(* IEC 61131-3 sources: generating_plc_code_with_llms/Code#2/ChatGPT_3.5/second run, 21 files *)

(* ---- 14.st ---- *)
// 7.18s
// 2
FUNCTION FC1001 :BOOL
VAR_INPUT
    MEW: REAL;
    SP: REAL;
    HYS: REAL;
END_VAR
VAR_IN_OUT
    OUT:BOOL;
END_VAR
VAR
    P_HYS: REAL;
END_VAR
    // Calculate the switching hysteresis as a percentage of the setpoint
    P_HYS := SP * HYS / 100.0;

    // Check if the measured value exceeds the upper threshold
    IF MEW > SP + P_HYS THEN
        OUT := TRUE;
    ELSIF MEW < SP - P_HYS THEN
        OUT := FALSE;
    END_IF;

    // Return the output status
    RETURN OUT;
END_FUNCTION

(* ---- 15.st ---- *)
// 8.77s
// 2
FUNCTION FC1002 :BOOL
VAR_INPUT
    E_A, SENSOR: BOOL;
    ZEITW: TIME;
END_VAR
VAR_IN_OUT
    ZEIT:TON;
    P_HU, P_AL: BOOL;
END_VAR
    // Check if the monitoring system is switched on
    IF E_A THEN
        // Reset the timer if the sensor reports an approach
        IF SENSOR THEN
            ZEIT(IN := FALSE);
        ELSE
            // Start the timer if the sensor doesn't report an approach
            ZEIT(IN := TRUE, PT := ZEITW);
        END_IF;

        // Check if the timer has reached the specified time
        IF ZEIT.Q THEN
            // Switch off the warning signal and turn on the alarm
            P_HU := FALSE;
            P_AL := TRUE;
        ELSE
            // Switch on the warning signal
            P_HU := SENSOR;
            // Turn off the alarm
            P_AL := FALSE;
        END_IF;
    ELSE
        // Switch off the monitoring system, warning signal, and alarm
        ZEIT(IN := FALSE);
        P_HU := FALSE;
        P_AL := FALSE;
    END_IF;

    // Return the switched on status of the monitoring system
    RETURN E_A;
END_FUNCTION

(* ---- 18.st ---- *)
// 6.77s
// 4
FUNCTION FC1003 : VOID
VAR_INPUT
    IN_R: REAL;
    IN_MAX, IN_MIN: REAL;
    OUT_MAX, OUT_MIN: REAL;
END_VAR
VAR_OUTPUT
    OUT_R: REAL;
    FEH: BOOL;
END_VAR
VAR_TEMP
    DIFF1, DIFF2: REAL;
END_VAR

IF (IN_MAX <> IN_MIN) THEN
    // Calculate the difference between the input and output ranges
    DIFF1 := OUT_MAX - OUT_MIN;
    DIFF2 := IN_MAX - IN_MIN;

    // Perform the range mapping
    OUT_R := OUT_MIN + ((IN_R - IN_MIN) / DIFF2) * DIFF1;

    // Check for out-of-range conditions
    IF (OUT_R < OUT_MIN) THEN
        OUT_R := OUT_MIN;
        FEH := TRUE;  // Set error flag
    ELSIF (OUT_R > OUT_MAX) THEN
        OUT_R := OUT_MAX;
        FEH := TRUE;  // Set error flag
    ELSE
        FEH := FALSE; // No error
    END_IF;
ELSE
    // Avoid division by zero if IN_MAX is equal to IN_MIN
    OUT_R := OUT_MIN;
    FEH := TRUE;  // Set error flag
END_IF;

(* ---- 19.st ---- *)
// 11.44s
// 2
FUNCTION_BLOCK FB1005
VAR_INPUT
    START: BOOL;
    DICKE, V_MAX, V_MIN: REAL;
END_VAR
VAR_OUTPUT
    D_MAX, D_MIN: REAL;
    P1: BOOL;
END_VAR
VAR
    FO: BOOL;
    M_MAX, M_MIN: REAL;
END_VAR
METHOD Messung : BOOL
    // Measure the thickness and update M_MAX, M_MIN
    M_MAX := MAX(M_MAX, DICKE);
    M_MIN := MIN(M_MIN, DICKE);

    // Check if the measured values are outside the tolerance band
    IF M_MAX > V_MAX OR M_MIN < V_MIN THEN
        P1 := TRUE;  // Turn on the reject light
    ELSE
        P1 := FALSE; // Turn off the reject light
    END_IF;

    // Return FALSE to end the measurement
    RETURN FALSE;
END_METHOD

METHOD StartMeasurement : BOOL
    // Start a new measurement cycle
    M_MAX := 0;
    M_MIN := 0;
    P1 := FALSE; // Turn off the reject light

    // Return TRUE to start the measurement
    RETURN TRUE;
END_METHOD

METHOD EndMeasurement : BOOL
    // Update output values with the results of the measurement
    D_MAX := M_MAX;
    D_MIN := M_MIN;

    // Return FALSE to end the measurement
    RETURN FALSE;
END_METHOD

METHOD FB1005 : BOOL
    // Check if the measurement is ongoing
    IF START THEN
        // If not in the measurement, start a new cycle
        IF NOT FO THEN
            FO := TRUE;
            RETURN StartMeasurement();
        // If already in the measurement, continue
        ELSE
            RETURN Messung();
        END_IF;
    // If the sensor is off, end the measurement
    ELSE
        IF FO THEN
            FO := FALSE;
            RETURN EndMeasurement();
        END_IF;
    END_IF;
END_METHOD
END_FUNCTION_BLOCK

(* ---- 20.st ---- *)
// 10.46s
// 2
FUNCTION_BLOCK INTERLOCK
VAR_INPUT
    I1: BOOL;
    I2: BOOL;
    TL: TIME;
END_VAR
VAR_OUTPUT
    Q1: BOOL;
    Q2: BOOL;
END_VAR
VAR
    T1: TOF;
    T2: TOF;
END_VAR

METHOD InterlockControl: BOOL
    // Control the interlock logic
    IF NOT T1.PT THEN
        // Start timer T1 when I1 is TRUE
        T1(IN := I1, PT := TL);
    ELSE
        // Reset timer T1 when I1 goes FALSE
        T1(IN := NOT I1);
    END_IF;

    IF NOT T2.PT THEN
        // Start timer T2 when I2 is TRUE
        T2(IN := I2, PT := TL);
    ELSE
        // Reset timer T2 when I2 goes FALSE
        T2(IN := NOT I2);
    END_IF;

    // Set Q1 only if T1 is not running and I1 is TRUE
    IF NOT T1.Q THEN
        Q1 := I1;
    END_IF;

    // Set Q2 only if T2 is not running and I2 is TRUE
    IF NOT T2.Q THEN
        Q2 := I2;
    END_IF;

    // Return TRUE to keep the method running
    RETURN TRUE;
END_METHOD

METHOD Initialize: BOOL
    // Reset timers and outputs at the beginning
    T1(IN := FALSE);
    T2(IN := FALSE);
    Q1 := FALSE;
    Q2 := FALSE;

    // Return FALSE to end the initialization
    RETURN FALSE;
END_METHOD

METHOD INTERLOCK: BOOL
    // Run the initialization at the start
    IF NOT T1.Q THEN
        RETURN Initialize();
    ELSE
        // Run the interlock control logic
        RETURN InterlockControl();
    END_IF;
END_METHOD
END_FUNCTION_BLOCK

(* ---- 21.st ---- *)
// 47.04s
// weiter generieren
// 2
FUNCTION_BLOCK BURNER
VAR_INPUT
    IN : BOOL;
    STAGE2 : BOOL;
    OVER_TEMP : BOOL;
    OIL_TEMP : BOOL := TRUE;
    FLAME : BOOL;
    RST : BOOL;
    RST_TIMER : BOOL;
    PRE_HEAT_TIME : TIME := t#5s;
    PRE_VENT_TIME : TIME := t#15s;
    PRE_IGNITE_TIME : TIME := t#15s;
    POST_IGNITE_TIME : TIME := t#25s;
    STAGE2_DELAY : TIME := t#10s;
    SAFETY_TIME : TIME := t#5s;
    LOCKOUT_TIME : TIME := t#10s;
    MULTIPLE_IGNITION : BOOL := TRUE;
    KW1 : REAL;
    KW2 : REAL;
END_VAR
VAR_OUTPUT
    MOTOR : BOOL;
    COIL1 : BOOL;
    COIL2 : BOOL;
    PRE_HEAT : BOOL;
    IGNITE : BOOL;
    FAIL : BOOL;
    KWH : REAL;
    STATUS : BYTE;
END_VAR
VAR_IN_OUT
    RUNTIME1 : UDINT;
    RUNTIME2 : UDINT;
    CYCLES : UDINT;
END_VAR
VAR
    state : INT;
    last : TIME;
    tx : TIME;
    last_change : TIME;
    timer1 : TON;
    timer2 : TON;
    oil_temp_last : BOOL;
    cycles2 : UDINT;
END_VAR

METHOD BurnerControl : BOOL
    tx := Tcyclic - last;
    last := Tcyclic;

    // Reset error flags
    FAIL := FALSE;

    // State machine for burner control
    CASE state OF
        110:
            // Standby - Wait for start signal
            IF IN THEN
                PRE_HEAT := TRUE;
                state := 111;  // Transition to startup sequence
            END_IF;
        111:
            // Startup Sequence
            IF (NOT OVER_TEMP) AND (NOT PRE_HEAT) THEN
                // Continue with startup sequence
                IF NOT OIL_TEMP THEN
                    IF timer1(IN := TRUE, PT := PRE_HEAT_TIME) THEN
                        // Fuel oil warming has not responded in time
                        STATUS := 1;
                        FAIL := TRUE;
                        state := 110;  // Return to standby
                    END_IF;
                ELSE
                    // Fuel oil warming responded, move to next step
                    MOTOR := TRUE;
                    COIL1 := TRUE;
                    timer1(IN := TRUE, PT := PRE_VENT_TIME);
                    state := 112;
                END_IF;
            END_IF;
        112:
            // Burner runs on stage 1
            IF timer1.Q THEN
                IGNITE := TRUE;
                COIL1 := FALSE;
                timer2(IN := TRUE, PT := PRE_IGNITE_TIME);
                state := 113;
            END_IF;
        113:
            // Burner runs on stage 2
            IF (STAGE2 AND timer2.Q) THEN
                COIL2 := TRUE;
            END_IF;
    END_CASE;

    // Check for errors during startup sequence
    IF (state = 112) AND FLAME THEN
        // Flame sensor is active during aeration
        STATUS := 2;
        FAIL := TRUE;
        state := 110;  // Return to standby
    END_IF;

    // Check for errors during burner operation
    IF (state = 113) AND (NOT FLAME) THEN
        IF timer2.Q THEN
            // No flame after specified time
            STATUS := 4;
            FAIL := TRUE;
            state := 110;  // Return to standby
        END_IF;

        // Check for multiple ignitions
        IF MULTIPLE_IGNITION AND FLAME AND (timer2.ET > 0) THEN
            IGNITE := TRUE;
            COIL2 := FALSE;
            cycles2 := cycles2 + 1;
            state := 113;
        END_IF;
    END_IF;

    // Boiler overheating protection
    IF OVER_TEMP THEN
        STATUS := 9;
        FAIL := TRUE;
        state := 110;  // Return to standby
    END_IF;

    // Lockout timer
    IF FAIL THEN
        IF NOT RST_TIMER THEN
            IF timer1.Q OR timer2.Q THEN
                timer1(IN := FALSE);
                timer2(IN := FALSE);
                timer1(IN := FALSE, PT := LOCKOUT_TIME);
                state := 110;  // Return to standby
            END_IF;
        END_IF;
    END_IF;

    // Update runtime and cycles
    IF state = 113 THEN
        RUNTIME1 := RUNTIME1 + tx;
    END_IF;

    // Update outputs
    KWH := (REAL)(cycles2 + (state = 113)) * KW2 + (REAL)CYCLES * KW1;
    CYCLES := cycles2 + (state = 113);

    RETURN state = 113;  // Return TRUE when the burner is running
END_METHOD;

METHOD BurnerStatus : VOID
    // Output the current status
    CASE state OF
        110: STATUS := 110;  // Standby
        111: STATUS := 111;  // Startup sequence is executed
        112: STATUS := 112;  // Burner runs on stage 1
        113: STATUS := 113;  // Burner runs on stage 2
    END_CASE;
END_METHOD;
END_FUNCTION_BLOCK

(* ---- 1.st ---- *)
// 4.91s
// 3
VAR
    xAllOn : BOOL;
    xAllOff : BOOL;

    xAlarm1 : BOOL;
    xAlarm2 : BOOL;
END_VAR

xAllOn := FALSE;
xAllOff := FALSE;
xAlarm1 := FALSE;
xAlarm2 := FALSE;

IF xAllOn THEN
    xAlarm1 := TRUE;
    xAlarm2 := TRUE;
    xAllOn := FALSE;
END_IF

IF xAllOff THEN
    xAlarm1 := FALSE;
    xAlarm2 := FALSE;
    xAllOff := FALSE;
END_IF

(* ---- 10.st ---- *)
// 4.44s
// 4
VAR_INPUT
    X : REAL;
END_VAR

VAR
    Y : REAL;
END_VAR

Y := 1 / (1 + EXP(-X));

(* ---- 11.st ---- *)
// 4.02s
// 4
VAR_INPUT
    x : REAL;
END_VAR

VAR
    result : INT;
END_VAR

IF x > 0 THEN
    result := 1;
ELSIF x < 0 THEN
    result := -1;
ELSE
    result := 0;
END_IF

(* ---- 12.st ---- *)
// 4.07s
// 4
VAR
    X : REAL;
    sinhX : REAL;
END_VAR

sinhX := (EXP(X) - EXP(-X)) / 2.0;

(* ---- 13.st ---- *)
// 5.81s
// 2
VAR CONSTANT
    MAXNUMBERS : UINT := 99;
END_VAR

VAR
    aNumbers : ARRAY[0..MAXNUMBERS] OF INT;
    nCnt : INT;
END_VAR

nCnt := 0;

REPEAT
    // Check if the current number is 10
    IF aNumbers[nCnt] = 10 THEN
        // Abort the search if 10 is found
        EXIT;
    END_IF;

    // Increment the counter
    nCnt := nCnt + 1;

    // Check if the end of the list is reached
    IF nCnt > MAXNUMBERS THEN
        // Abort if the end of the list is reached without finding 10
        EXIT;
    END_IF;
UNTIL FALSE;

(* ---- 16.st ---- *)
// 10.51s
// 2
VAR
    North_green : BOOL;
    North_yellow : BOOL;
    North_red : BOOL;
    East_green : BOOL;
    East_yellow : BOOL;
    East_red : BOOL;
    T1 : TON;
END_VAR

T1(IN := TRUE, PT := T#5000ms);  // Timer T1 for the overall cycle

IF T1.Q THEN
    // Between 0ms and 5000ms
    North_green := TRUE;
    North_yellow := FALSE;
    North_red := FALSE;
    East_green := FALSE;
    East_yellow := FALSE;
    East_red := TRUE;
ELSE
    // After 5000ms
    North_green := FALSE;
    North_yellow := TRUE;
    North_red := FALSE;
    East_green := FALSE;
    East_yellow := FALSE;
    East_red := TRUE;
END_IF;

IF NOT T1.Q AND T1.ET THEN
    // Between 5500ms and 9500ms
    North_green := FALSE;
    North_yellow := FALSE;
    North_red := TRUE;
    East_green := TRUE;
    East_yellow := FALSE;
    East_red := FALSE;
END_IF;

IF NOT T1.Q AND T1.ETT THEN
    // Between 9500ms and 10000ms
    North_green := FALSE;
    North_yellow := FALSE;
    North_red := TRUE;
    East_green := FALSE;
    East_yellow := TRUE;
    East_red := FALSE;
END_IF;

(* ---- 17.st ---- *)
// 7.22s
// 4
VAR
    aiOutside : INT;
    aiHumidity: INT;
    sShowText : STRING[80];
END_VAR

// Read temperature and humidity values (replace with actual input values)
aiOutside := ...;
aiHumidity := ...;

// Evaluate temperature
IF aiOutside < 18 THEN
    sShowText := 'Cold';
ELSIF aiOutside >= 18 AND aiOutside <= 25 THEN
    // Evaluate humidity within the nested IF
    IF aiHumidity >= 40 AND aiHumidity <= 75 THEN
        sShowText := 'Opt';
    ELSE
        sShowText := 'Temp. OK';
    END_IF;
ELSE
    sShowText := 'Hot';
END_IF;

(* ---- 2.st ---- *)
// 4.61s
// 4
VAR_INPUT
    N : INT;
    K : INT;
    i : INT;
END_VAR

VAR
    result : INT;
    numerator : INT;
    denominator : INT;
END_VAR

result := 0;
numerator := 1;
denominator := 1;

IF K >= 0 AND K <= N THEN
    FOR i := 1 TO K DO
        numerator := numerator * (N - i + 1);
        denominator := denominator * i;
    END_FOR

    result := numerator / denominator;
END_IF

(* ---- 3.st ---- *)
// 4.94s
// 2
VAR_INPUT
    X : INT;
END_VAR

VAR
    t1 : DINT;
    t2 : DINT;
    x_tmp : INT;
END_VAR

t1 := 0;
t2 := 1;

IF X = 0 THEN
    x_tmp := t1;
ELSIF X = 1 THEN
    x_tmp := t2;
ELSE
    FOR i := 2 TO X DO
        x_tmp := t1 + t2;
        t1 := t2;
        t2 := x_tmp;
    END_FOR
END_IF

(* ---- 4.st ---- *)
// 7.06s
// 2
VAR
    aiLevel : INT;
    PercentLevel : UINT;
    doLow : BOOL;
    doOk : BOOL;
    doHigh : BOOL;
    doAlarm : BOOL;
END_VAR

aiLevel := ... // Read the analog input level (0 - 32767) from your system

// Convert analog input to percentage (0 - 100%)
PercentLevel := UINT_TO(aiLevel * 100 / 32767);

CASE PercentLevel OF
    (PercentLevel < 1):
        doLow := TRUE;
        doOk := FALSE;
        doHigh := FALSE;
        doAlarm := TRUE; // Activate the warning horn
    (PercentLevel >= 1 AND PercentLevel <= 75):
        doLow := FALSE;
        doOk := TRUE;
        doHigh := FALSE;
        doAlarm := FALSE;
    (PercentLevel > 75):
        doLow := FALSE;
        doOk := FALSE;
        doHigh := TRUE;
        doAlarm := FALSE;
END_CASE

(* ---- 5.st ---- *)
// 7.51s
// 3
VAR
    Start_Loop : BOOL := FALSE;
    one_hour : TIME := T#1h;
    One_Hour_Timer : TON;
    Gate_Open : BOOL := FALSE;
    Close_Gate_Inst : BOOL := FALSE;
    Sensed_Car : BOOL := FALSE;
    Sensed_Car_Inst : BOOL := FALSE;
    Sensed_App : BOOL := FALSE;
    Mobile_Inst : BOOL := FALSE;
    Auth : STRING;
    my_defined_str : STRING := 'abcd';
END_VAR

// Main control logic
IF NOT Start_Loop THEN
    // Start the one-hour timer when Start_Loop is FALSE
    One_Hour_Timer(IN := NOT Gate_Open AND NOT Close_Gate_Inst, PT := one_hour);

    // Check if the timer timed out
    IF One_Hour_Timer.Q THEN
        Close_Gate_Inst := TRUE;
    END_IF;

    // Check for sensed car or app with matching Auth string
    IF (Sensed_Car AND NOT Sensed_Car_Inst) OR (Sensed_App AND Mobile_Inst AND Auth = my_defined_str) THEN
        Gate_Open := TRUE;
        Close_Gate_Inst := FALSE;
    END_IF;

    // Reset the timer if the gate is open
    IF Gate_Open THEN
        One_Hour_Timer(IN := FALSE);
    END_IF;
ELSE
    // Reset the timer when Start_Loop is TRUE
    One_Hour_Timer(IN := FALSE);
    Close_Gate_Inst := FALSE;
    Gate_Open := FALSE;
END_IF

(* ---- 6.st ---- *)
// 12.6s
// 4
VAR CONSTANT
    WAIT : UINT:= 0;
    TOP_POSITION : UINT:= 1;
    BOTTOM_POSITION : UINT:= 2;
    GETBOX : UINT:= 3;
    UNLOAD_POSITION : UINT:= 4;
    UNLOAD_BOX : UINT:= 5;
END_VAR

VAR
    doConvTop: BOOL;
    doConvBottom: BOOL;
    doConvLift: BOOL;
    doLiftTop: BOOL;
    doLiftBottom: BOOL;
    doLiftUnload: BOOL;
    diConvTop: BOOL;
    diConvBottom: BOOL;
    diLiftTop: BOOL;
    diLiftBottom: BOOL;
    diLiftUnload: BOOL;
    diBoxLift: BOOL;
    selectLift: UINT;
    ConvTopOn: BOOL;
    ConvBottomOn: BOOL;
END_VAR

CASE selectLift OF
    WAIT:
        // Check if either light barrier is activated
        IF diConvTop THEN
            doConvTop := FALSE;
            ConvTopOn := FALSE;
            selectLift := TOP_POSITION;
        ELSIF diConvBottom THEN
            doConvBottom := FALSE;
            ConvBottomOn := FALSE;
            selectLift := BOTTOM_POSITION;
        END_IF;
        // Reset lift control signals
        doLiftTop := FALSE;
        doLiftBottom := FALSE;
        doLiftUnload := FALSE;
    TOP_POSITION:
        // Move lift to top position
        doLiftTop := TRUE;
        IF diLiftTop THEN
            doLiftTop := FALSE;
            selectLift := GETBOX;
        END_IF;
    BOTTOM_POSITION:
        // Move lift to bottom position
        doLiftBottom := TRUE;
        IF diLiftBottom THEN
            doLiftBottom := FALSE;
            selectLift := GETBOX;
        END_IF;
    GETBOX:
        // Activate lift conveyor until crate is at lift
        doConvLift := TRUE;
        IF diBoxLift THEN
            doConvLift := FALSE;
            selectLift := UNLOAD_POSITION;
        END_IF;
    UNLOAD_POSITION:
        // Move lift to unload position
        doLiftUnload := TRUE;
        IF diLiftUnload THEN
            doLiftUnload := FALSE;
            selectLift := UNLOAD_BOX;
        END_IF;
    UNLOAD_BOX:
        // Unload box onto the unloading conveyor
        // Once the box has left the lift, it's ready for the next request
        IF NOT diBoxLift THEN
            selectLift := WAIT;
        END_IF;
END_CASE;

(* ---- 7.st ---- *)
// 5.63s
// 2
VAR CONSTANT
    MAX_INDEX: USINT := 4;
END_VAR

VAR
    aWeights : ARRAY[0..MAX_INDEX] OF INT;
    iCnt : USINT;
    sumWeight : DINT;
    avgWeight : INT;
END_VAR

sumWeight := 0;

FOR iCnt := 0 TO MAX_INDEX DO
    // Read individual loads from analog inputs (replace with actual input values)
    aWeights[iCnt] := ...;
    sumWeight := sumWeight + aWeights[iCnt];
END_FOR

// Calculate average weight
IF MAX_INDEX > 0 THEN
    avgWeight := sumWeight / (MAX_INDEX + 1);
ELSE
    avgWeight := 0; // To avoid division by zero
END_IF

(* ---- 8.st ---- *)
// 7.08s
// 2
VAR_INPUT
    X : REAL;
END_VAR

VAR
    w : REAL;
    i : INT;
    we : REAL;
    w1e : REAL;
    ewx : REAL;
    last : DWORD;
END_VAR

w := 0.0;
i := 0;
we := 0.0;
w1e := 0.0;

FOR i := 0 TO 1000 DO
    ewx := EXP(w * we);
    last := TIME();
    w := w - (w * we - X) / (we * (w + 1));
    IF ABS(ewx - EXP(w * we)) < 1.0E-9 OR ABS(TIME() - last) < T#1ms THEN
        EXIT; // Exit loop if convergence or max iterations reached
    END_IF;
END_FOR

(* ---- 9.st ---- *)
// 5.72s
// 2
VAR
    YEAR : INT;
END_VAR

IF (YEAR MOD 4 = 0 AND YEAR MOD 100 <> 0) OR (YEAR MOD 400 = 0) THEN
    // Leap year conditions:
    // - If divisible by 4 but not by 100
    // - If divisible by 400
    // It is a leap year
    // Implement your logic for a leap year here, e.g., set a variable or perform specific actions
ELSE
    // Not a leap year
    // Implement your logic for a non-leap year here, if needed
END_IF
